FUNCTION F_LogA3 
VAR_INPUT
	eLogLevel		: E_LogLevel;
	sMessage		: T_MaxString;
	aArg1			: ANY;
	aArg2			: ANY;
	aArg3			: ANY;
END_VAR

F_LogLA3(eLogLevel, Const.sGlobalLogger, sMessage, aArg1, aArg2, aArg3);

END_FUNCTION

(* stored: Version 1.1.0.1, ProductVersion 3.1.4024.6
   POU F_LogA3: Id {e7f0957a-d6ba-4de1-8a25-abd1924486df}, SpecialFunc None *)
